(* IEC 61131-3 sources: pandora/pandora/aws-platform-main/aws-platform-main/src/Motion, 6 files *)

(* ---- Axis.st ---- *)
USING Esab.Utils.Assets;

NAMESPACE Esab.Motion

    /// Interface defining an axis.
    /// The interface supports both linear and rotary axes, defined through hardware configuration.
    INTERFACE IAxis
        METHOD PowerOn
        END_METHOD

        METHOD PowerOff
        END_METHOD

        METHOD Reset
            VAR_INPUT
                Restart : BOOL;
            END_VAR
        END_METHOD

        METHOD ExecutePositioningCommand : AxisCommandError
            VAR_INPUT
                command : AxisPositioningCommand;
            END_VAR
        END_METHOD

        METHOD ExecuteHomingCommand : AxisCommandError
            VAR_INPUT
                command: AxisHomingCommand;
            END_VAR
        END_METHOD

        METHOD InvalidateHoming
        END_METHOD

        METHOD Halt
        END_METHOD

        METHOD SetJogSpeed
            VAR_INPUT
                value : LREAL;
            END_VAR
        END_METHOD

        METHOD SetJogHighSpeed
            VAR_INPUT
                value : LREAL;
            END_VAR
        END_METHOD

        METHOD SetObjectRadius
            VAR_INPUT
                value : LREAL;
            END_VAR
        END_METHOD

        METHOD JogPositive
            VAR_INPUT
                highSpeed : BOOL := FALSE;
            END_VAR
        END_METHOD

        METHOD JogNegative
            VAR_INPUT
                highSpeed : BOOL := FALSE;
            END_VAR
        END_METHOD

        METHOD IsEnabled : BOOL
        END_METHOD

        METHOD IsBusy : BOOL
        END_METHOD

        METHOD IsHomed : BOOL
        END_METHOD

        METHOD HasError : BOOL
        END_METHOD

        METHOD AtStandstill : BOOL
        END_METHOD

        METHOD ActualLinearPosition : LREAL
        END_METHOD

        METHOD ActualLinearVelocity : LREAL
        END_METHOD

        METHOD ActualAngularPosition : LREAL
        END_METHOD

        METHOD ActualAngularVelocity : LREAL
        END_METHOD
    END_INTERFACE

    TYPE
        AxisCommandError : INT(
            NoError := 0,
            UnsupportedCommandType := 1,
            UnsupportedHomingType := 2,
            AxisNotEnabled := 3
        ) := AxisCommandError#NoError;

        AxisPositioningCommand : STRUCT
            CommandType : AxisCommandType := AxisCommandType#Absolute;
            /// NOTE: Only modulo axes supports setting the mode.
            PositioningDirection : AxisPositioningDirection := AxisPositioningDirection#Nearest;
            Id : INT := 0;
            Position : LREAL := 0.0;
            Velocity : LREAL := -1.0;
            Acceleration : LREAL := -1.0;
            Deceleration : LREAL := -1.0;
            Jerk : LREAL := -1.0;
        END_STRUCT;

        AxisCommandType : INT(
            Invalid     := -1,
            Absolute    := 0,
            Relative    := 1,
            Velocity    := 2,
            Halt        := 3
        ) := AxisCommandType#Invalid;

        AxisPositioningDirection : INT(
            Nearest := 0,
            Positive := 1,
            Negative := 2
        ) := AxisPositioningDirection#Nearest;

        AxisHomingCommand : STRUCT
            HomingType : AxisHomingType := AxisHomingType#DirectAbsolute;
            Position : LREAL := 0.0;
        END_STRUCT;

        AxisHomingType : INT(
            Invalid := -1,
            DirectAbsolute := 0,
            DirectRelative := 1,
            Active := 2,
            Passive := 3,
            AbsoluteEncoderAdjustementRelative := 4,
            AbsoluteEncoderAdjustementAbsolute := 5
        ) := AxisHomingType#Invalid;

        AxisState : INT(
            Enabled := 0,
            Disabled := 1,
            Error := 2,
            Homing := 3,
            Moving := 4
        ) := AxisState#Disabled;

        AxisType : INT(
            Linear := 0,
            Rotary := 1
        ) := AxisType#Rotary;

        AxisRuntimeParameters : STRUCT
            JogSpeed : LREAL := 10.0;
            JogHighSpeed : LREAL := 20.0;
            ObjectRadius : LREAL := 1500.0;
        END_STRUCT;

        AxisHardwareConfiguration : STRUCT
            AxisType : AxisType := AxisType#Linear;
        END_STRUCT;
    END_TYPE

    CLASS AxisObservable IMPLEMENTS IAssetObservable
        VAR PUBLIC
            State : AxisState;
            Enabled : BOOL;
            Accelerating : BOOL;
            Decelerating : BOOL;
            Standstill : BOOL;
            Homed : BOOL;
            Error : BOOL;
            ErrorId : WORD;
            Busy : BOOL;
            Done : BOOL;
            LatestCommandId : INT;
            LinearPosition : LREAL;
            LinearVelocity : LREAL;
            AngularPosition : LREAL;
            AngularVelocity : LREAL;
            ObjectRadius : LREAL;
        END_VAR
    END_CLASS

END_NAMESPACE

(* ---- WeldHeadManipulator.st ---- *)
USING Esab.Hmi.Modules;
USING Esab.Utils.Assets;
USING Esab.Utils.Alarming;
USING System.FastMath;

NAMESPACE Esab.Motion

    INTERFACE IWeldHeadManipulator
        METHOD Enable : WeldHeadManipulatorErrorCode
        END_METHOD

        METHOD Disable
        END_METHOD

        /// Interpolated motion, axes will arrive at the same time
        METHOD Move : WeldHeadManipulatorErrorCode
            VAR_INPUT
                position : ARRAY [0..1] OF LREAL := [0.0, 0.0];
                speed : LREAL := -1;
            END_VAR
        END_METHOD

        /// Non-interpolated movement
        METHOD Move : WeldHeadManipulatorErrorCode
            VAR_INPUT
                position : ARRAY [0..1] OF LREAL := [0.0, 0.0];
                speed : ARRAY [0..1] OF LREAL := [-1.0, -1.0];
            END_VAR
        END_METHOD

        METHOD IsEnabled : BOOL
        END_METHOD

        METHOD GetPosition : ARRAY [0..1] OF LREAL
        END_METHOD

        METHOD GetSpeed : LREAL
        END_METHOD

        METHOD GetVelocity : ARRAY [0..1] OF LREAL
        END_METHOD

        METHOD GetControlMode : WeldHeadManipulatorControlMode
        END_METHOD

        METHOD SetControlMode
            VAR_INPUT
                controlMode : WeldHeadManipulatorControlMode;
            END_VAR
        END_METHOD
    END_INTERFACE

    /// Class that wraps all axes that are used to manipulate the welding head.
    /// Depending on the hardware configuration this may include:
    /// - Horizontal slide axis
    /// - Vertical slide axis
    /// - Tilt (Not implemented)
    /// - Clock position slide (Not implemented)
    CLASS WeldHeadManipulator EXTENDS Asset IMPLEMENTS IAssetRequester, IWeldHeadManipulator, IPositionChangedListener
        VAR PRIVATE
            _runtimeParameters : REF_TO WeldHeadManipulatorRuntimeParameters;
            _hardwareConfiguration : REF_TO WeldHeadManipulatorHardwareConfiguration;
            _assetsManager : IAssetsManager;

            _horizontalSlide : IAxis;
            _verticalSlide : IAxis;

            _horizontalSlideObservable : REF_TO AxisObservable;
            _verticalSlideObservable : REF_TO AxisObservable;

            _horizontalSlideCommand : Esab.Motion.AxisPositioningCommand;
            _verticalSlideCommand : Esab.Motion.AxisPositioningCommand;

            _currentJogDirection : JoystickPosition := JoystickPosition#None;
            _motionJoystick : IJoystick := NULL;
        END_VAR

        METHOD PUBLIC Setup
            VAR_INPUT
                runtimeParameters : REF_TO WeldHeadManipulatorRuntimeParameters;
                hardwareConfiguration : REF_TO WeldHeadManipulatorHardwareConfiguration;
                assetsManager : IAssetsManager;
                setupAlarm : IAlarm;
            END_VAR

            _runtimeParameters := runtimeParameters;
            _hardwareConfiguration := hardwareConfiguration;
            _assetsManager := assetsManager;

            _isSetup := _runtimeParameters <> NULL AND _hardwareConfiguration <> NULL AND _assetsManager <> NULL;
        END_METHOD

        METHOD PUBLIC OVERRIDE Execute
            SUPER.Execute();

            IF _setupAlarm.IsActive() THEN
                RETURN;
            END_IF;

            THIS.RequestMotionJoystick();

            IF _horizontalSlideObservable = NULL THEN
                _horizontalSlideObservable ?= _assetsManager.ObserveAsset(Esab.AssetIdentifier#HorizontalSlideAxis);
            END_IF;

            IF _verticalSlideObservable = NULL THEN
                _verticalSlideObservable ?= _assetsManager.ObserveAsset(Esab.AssetIdentifier#VerticalSlideAxis);
            END_IF;

            IF _runtimeParameters^.controlMode = WeldHeadManipulatorControlMode#JoystickJog THEN
                THIS.HandleSlideJog();
            END_IF;
        END_METHOD

        METHOD PUBLIC Enable : WeldHeadManipulatorErrorCode
            VAR_TEMP
                currentPosition : ARRAY [0..1] OF LREAL;
            END_VAR

            IF NOT THIS.RequestAndLockAxis() THEN
                Enable := WeldHeadManipulatorErrorCode#AssetsNotAvailable;
                RETURN;
            END_IF;

            IF NOT _horizontalSlide.IsEnabled() THEN
                _horizontalSlide.PowerOn();
            END_IF;

            IF NOT _verticalSlide.IsEnabled() THEN
                _verticalSlide.PowerOn();
            END_IF;

            IF _horizontalSlide.HasError() OR _verticalSlide.HasError() THEN
                Enable := WeldHeadManipulatorErrorCode#AxisError;
                RETURN;
            END_IF;

            currentPosition[0] := _horizontalSlide.ActualLinearPosition();
            currentPosition[1] := _verticalSlide.ActualLinearPosition();

            THIS.Move(currentPosition, -1.0);
        END_METHOD

        METHOD PUBLIC Disable
            IF _horizontalSlide <> NULL THEN
                _horizontalSlide.Halt();
            END_IF;

            IF _verticalSlide <> NULL THEN
                _verticalSlide.Halt();
            END_IF;

            THIS.UnlockAxis();
        END_METHOD

        METHOD PUBLIC Move : WeldHeadManipulatorErrorCode
            VAR_INPUT
                position : ARRAY [0..1] OF LREAL := [0.0, 0.0];
                speed : LREAL := -1;
            END_VAR

            VAR_TEMP
                speedComponents : ARRAY [0..1] OF LREAL;
                currentPosition : ARRAY [0..1] OF LREAL;
            END_VAR

            IF _horizontalSlide = NULL OR _verticalSlide = NULL THEN
                Move := WeldHeadManipulatorErrorCode#AssetsNotAvailable;
                RETURN;
            END_IF;

            IF _horizontalSlide.HasError() OR _verticalSlide.HasError() THEN
                Move := WeldHeadManipulatorErrorCode#AxisError;
                RETURN;
            END_IF;

            currentPosition[0] := _horizontalSlide.ActualLinearPosition();
            currentPosition[1] := _verticalSlide.ActualLinearPosition();

            IF speed > 1.0 THEN
                speedComponents := THIS.CalculateSpeed(speed, currentPosition, position);
            ELSIF speed < 0.0 THEN
                speedComponents := THIS.CalculateSpeed(_runtimeParameters^.defaultSpeed, currentPosition, position);
            ELSE
                Move := WeldHeadManipulatorErrorCode#SpeedSetTooLow;
                RETURN;
            END_IF;

            _horizontalSlideCommand.CommandType := AxisCommandType#Absolute;
            _horizontalSlideCommand.Velocity := speedComponents[0];
            _horizontalSlideCommand.Position := position[0];

            _verticalSlideCommand.CommandType := AxisCommandType#Absolute;
            _verticalSlideCommand.Velocity := speedComponents[1];
            _verticalSlideCommand.Position := position[1];

            _horizontalSlide.ExecutePositioningCommand(_horizontalSlideCommand);
            _verticalSlide.ExecutePositioningCommand(_verticalSlideCommand);
        END_METHOD

        METHOD PUBLIC Move : WeldHeadManipulatorErrorCode
            VAR_INPUT
                position : ARRAY [0..1] OF LREAL := [0.0, 0.0];
                speed : ARRAY [0..1] OF LREAL := [-1.0, -1.0];
            END_VAR

            VAR_TEMP
                speedComponents : ARRAY [0..1] OF LREAL;
            END_VAR

            IF _horizontalSlide = NULL OR _verticalSlide = NULL THEN
                Move := WeldHeadManipulatorErrorCode#AssetsNotAvailable;
                RETURN;
            END_IF;

            IF _horizontalSlide.HasError() OR _verticalSlide.HasError() THEN
                Move := WeldHeadManipulatorErrorCode#AxisError;
                RETURN;
            END_IF;

            IF _runtimeParameters^.controlMode <> WeldHeadManipulatorControlMode#MoveToPosition THEN
                Move := WeldHeadManipulatorErrorCode#IncorrectControlMode;
                RETURN;
            END_IF;

            speedComponents := speed;

            _horizontalSlideCommand.CommandType := AxisCommandType#Absolute;
            _horizontalSlideCommand.Velocity := speedComponents[0];
            _horizontalSlideCommand.Position := position[0];

            _verticalSlideCommand.CommandType := AxisCommandType#Absolute;
            _verticalSlideCommand.Velocity := speedComponents[1];
            _verticalSlideCommand.Position := position[1];

            _horizontalSlide.ExecutePositioningCommand(_horizontalSlideCommand);
            _verticalSlide.ExecutePositioningCommand(_verticalSlideCommand);
        END_METHOD

        METHOD PUBLIC IsEnabled : BOOL
            IF THIS.InControl() THEN
                IsEnabled := _horizontalSlide.IsEnabled() AND _verticalSlide.IsEnabled();
            ELSE
                IsEnabled := FALSE;
            END_IF;
        END_METHOD

        METHOD PUBLIC GetPosition : ARRAY [0..1] OF LREAL
            IF _horizontalSlideObservable <> NULL AND _verticalSlideObservable <> NULL THEN
                GetPosition[0] := _horizontalSlideObservable^.LinearPosition;
                GetPosition[1] := _verticalSlideObservable^.LinearPosition;
            END_IF;
        END_METHOD

        METHOD PUBLIC GetSpeed : LREAL
            IF _horizontalSlideObservable <> NULL AND _verticalSlideObservable <> NULL THEN
                GetSpeed := Sqrt(_horizontalSlideObservable^.LinearVelocity * _horizontalSlideObservable^.LinearVelocity +
                                 _verticalSlideObservable^.LinearVelocity * _verticalSlideObservable^.LinearVelocity);
            END_IF;
        END_METHOD

        METHOD PUBLIC GetVelocity : ARRAY [0..1] OF LREAL
            IF _horizontalSlideObservable <> NULL AND _verticalSlideObservable <> NULL THEN
                GetVelocity[0] := _horizontalSlideObservable^.LinearVelocity;
                GetVelocity[1] := _verticalSlideObservable^.LinearVelocity;
            END_IF;
        END_METHOD

        METHOD PUBLIC GetControlMode : WeldHeadManipulatorControlMode
            GetControlMode := _runtimeParameters^.controlMode;
        END_METHOD

        METHOD PUBLIC SetControlMode
            VAR_INPUT
                controlMode : WeldHeadManipulatorControlMode;
            END_VAR;

            IF controlMode <> WeldHeadManipulatorControlMode#JoystickJog THEN
                _currentJogDirection := JoystickPosition#None;
            END_IF;

            _runtimeParameters^.controlMode := controlMode;
        END_METHOD

        METHOD PUBLIC AssetAssigned
            VAR_INPUT
                asset : REF_TO Esab.Utils.Assets.Asset;
            END_VAR

            ;
        END_METHOD

        METHOD PUBLIC AssetRemoved
            VAR_INPUT
                identifier : INT;
            END_VAR

            ;
        END_METHOD

        METHOD PUBLIC OVERRIDE Observe : IAssetObservable
            ;
        END_METHOD

        METHOD PRIVATE RequestAndLockAxis : BOOL
            VAR_TEMP
                success : BOOL := TRUE;
                asset : REF_TO Asset := NULL;
            END_VAR

            IF _hardwareConfiguration^.horizontalSlideAxis AND _horizontalSlide = NULL THEN
                asset := _assetsManager.RequestAssetHandle(THIS, Esab.AssetIdentifier#HorizontalSlideAxis);
                IF asset <> NULL THEN
                    _horizontalSlide ?= asset^;
                ELSE
                    success := FALSE;
                END_IF;
            END_IF;

            IF _hardwareConfiguration^.verticalSlideAxis AND _verticalSlide = NULL THEN
                asset := _assetsManager.RequestAssetHandle(THIS, Esab.AssetIdentifier#VerticalSlideAxis);
                IF asset <> NULL THEN
                    _verticalSlide ?= asset^;
                ELSE
                    success := FALSE;
                END_IF;
            END_IF;

            IF success THEN
                IF _horizontalSlide <> NULL THEN
                    asset ?= _horizontalSlide;
                    asset^.Lock();
                END_IF;

                IF _verticalSlide <> NULL THEN
                    asset ?= _verticalSlide;
                    asset^.Lock();
                END_IF;
            END_IF;

            RequestAndLockAxis := success;
        END_METHOD

        METHOD PRIVATE InControl : BOOL
            VAR_TEMP
                asset : REF_TO asset;
            END_VAR

            InControl := TRUE;

            IF _horizontalSlide <> NULL THEN
                asset ?= _horizontalSlide;
                IF NOT asset^.IsLocked() THEN
                    InControl := FALSE;
                END_IF;
            ELSE
                InControl := FALSE;
            END_IF;

            IF _verticalSlide <> NULL THEN
                asset ?= _verticalSlide;
                IF NOT asset^.IsLocked() THEN
                    InControl := FALSE;
                END_IF;
            ELSE
                InControl := FALSE;
            END_IF;
        END_METHOD

        METHOD PRIVATE UnlockAxis
            VAR_TEMP
                asset : REF_TO Asset;
            END_VAR

            IF _horizontalSlide <> NULL THEN
                asset ?= _horizontalSlide;
                asset^.Unlock();
            END_IF;

            IF _verticalSlide <> NULL THEN
                asset ?= _verticalSlide;
                asset^.Unlock();
            END_IF;
        END_METHOD

        METHOD PRIVATE CalculateSpeed : ARRAY [0..1] OF LREAL
            VAR_INPUT
                speed : LREAL;
                currentPosition : ARRAY [0..1] OF LREAL;
                targetPosition : ARRAY [0..1] OF LREAL;
            END_VAR

            VAR_TEMP
                theta : LREAL;
                distance : ARRAY [0..1] OF LREAL;
            END_VAR

            distance[0] := Abs(targetPosition[0]-currentPosition[0]);
            distance[1] := Abs(targetPosition[1]-currentPosition[1]);

            theta := ATan(distance[1] / distance[0]);

            CalculateSpeed[0] := speed * Cos(theta);
            CalculateSpeed[1] := speed * Sin(theta);

            IF CalculateSpeed[0] < 1.0 THEN
                CalculateSpeed[0] := 1.0;
            END_IF;

            IF CalculateSpeed[1] < 1.0 THEN
                CalculateSpeed[1] := 1.0;
            END_IF;
        END_METHOD

        METHOD PUBLIC OnPositionChanged
            VAR_INPUT
                position : JoystickPosition;
            END_VAR
                IF _runtimeParameters^.controlMode <> WeldHeadManipulatorControlMode#JoystickJog THEN
                    RETURN;
                END_IF;

                _currentJogDirection := position;
        END_METHOD

        METHOD PRIVATE HandleSlideJog
            IF _horizontalSlide = NULL OR _verticalSlide = NULL THEN
                RETURN;
            END_IF;

            IF _horizontalSlide.HasError() OR _verticalSlide.HasError() THEN
                RETURN;
            END_IF;

            CASE _currentJogDirection OF
                JoystickPosition#None:
                    _horizontalSlide.Halt();
                    _verticalSlide.Halt();
                JoystickPosition#Center:
                    _horizontalSlide.Halt();
                    _verticalSlide.Halt();
                JoystickPosition#Up:
                    _horizontalSlide.Halt();
                    _verticalSlide.JogPositive();
                JoystickPosition#Down:
                    _horizontalSlide.Halt();
                    _verticalSlide.JogNegative();
                JoystickPosition#Square:
                    _horizontalSlide.JogPositive();
                    _verticalSlide.Halt();
                JoystickPosition#Triangle:
                    _horizontalSlide.JogNegative();
                    _verticalSlide.Halt();
            END_CASE;
        END_METHOD

        METHOD PRIVATE RequestMotionJoystick
            VAR_TEMP
                assetHandle : REF_TO Asset;
            END_VAR

            IF _motionJoystick = NULL THEN
                assetHandle := THIS._assetsManager.RequestAssetHandle(THIS, Esab.AssetIdentifier#P_Joystick_MotionJoystick);

                IF assetHandle <> NULL THEN
                    _motionJoystick ?= assetHandle^;
                    IF _motionJoystick <> NULL THEN
                        _motionJoystick.SetPositionChangedListener(THIS);
                    END_IF;
                END_IF;
            END_IF;
        END_METHOD

    END_CLASS

    TYPE
        WeldHeadManipulatorRuntimeParameters : STRUCT
        /// Speed used when move command speed < 0.0
            defaultSpeed : LREAL := 10.0;
            controlMode : WeldHeadManipulatorControlMode;
        END_STRUCT;

        WeldHeadManipulatorHardwareConfiguration : STRUCT
            /// X-axis
            horizontalSlideAxis : BOOL := TRUE;
            /// Z-axis
            verticalSlideAxis : BOOL := TRUE;
        END_STRUCT;

        WeldHeadManipulatorErrorCode : INT(
            NoError := 0,
            AssetsNotAvailable := 1,
            AxisError := 2,
            SpeedSetTooLow := 3,
            IncorrectControlMode := 4
        ) := WeldHeadManipulatorErrorCode#NoError;

        WeldHeadManipulatorControlMode : INT(
            NoControl := 0,
            JoystickJog := 1,
            MoveToPosition := 2
        ) := WeldHeadManipulatorControlMode#NoControl;
    END_TYPE
END_NAMESPACE

(* ---- AnalogAxis.st ---- *)
USING Esab.Motion.MeasurementSystem;
USING Esab.Utils.Assets;
USING Esab.Utils.Timer;
USING Esab.Utils.Alarming;
USING Esab.Io;

USING System.FastMath;

NAMESPACE Esab.Motion

    /// Implements an axis with the following properties:
    ///     - The axis is controlled via digital and analog I/O:
    ///         - Forwards/positive direction (digital out)
    ///         - Backwards/negative direction (digital out)
    ///         - Speed (analog out)
    /// To measure the position (if applicable) a measurement system should
    /// be provided. The axis will work "fine" without it but it will be limited to
    /// speed control without feedback.
    CLASS AnalogAxis EXTENDS Asset IMPLEMENTS IAxis, IMeasurementSystemListener
        VAR PRIVATE
            _io : REF_TO AnalogAxisIo;
            _runtimeParameters : REF_TO AnalogAxisRuntimeParameters;
            _hardwareConfiguration : REF_TO AnalogAxisHardwareConfiguration;
            _measurementSystem : IMeasurementSystem1D;
            _speedMeasurementTimer : ITimer;
            _speedMonitoringAlarm : IAlarm;

            _observable : AxisObservable;

            _setVelocity : LREAL := 0.0;
            _jogPositive : BOOL := FALSE;
            _jogNegative : BOOL := FALSE;
            _highSpeed : BOOL := FALSE;
            _isJogging : BOOL := FALSE;
            _isHomed : BOOL := FALSE;
            _poweredOn : BOOL := FALSE;
            _measuring : BOOL := FALSE;
            _hasPassedReferencePointOnce : BOOL := FALSE;
        END_VAR

        METHOD PUBLIC Setup
            VAR_INPUT
                io : REF_TO AnalogAxisIo;
                runtimeParameters : REF_TO AnalogAxisRuntimeParameters;
                hardwareConfiguration : REF_TO AnalogAxisHardwareConfiguration;
                measurementSystem : IMeasurementSystem1D;
                speedMeasurementTimer : ITimer;
                speedMonitoringAlarm : IAlarm;
                setupAlarm : IAlarm;
            END_VAR

            _io := io;
            _runtimeParameters := runtimeParameters;
            _hardwareConfiguration := hardwareConfiguration;
            _measurementSystem := measurementSystem;
            _speedMeasurementTimer := speedMeasurementTimer;
            _speedMonitoringAlarm := speedMonitoringAlarm;
            _setupAlarm := setupAlarm;

            _isSetup := _io <> NULL AND
                        _hardwareConfiguration <> NULL AND
                        _runtimeParameters <> NULL AND
                        _measurementSystem <> NULL AND
                        _speedMonitoringAlarm <> NULL;

            IF _isSetup THEN
                _measurementSystem.SetListener(THIS);
            END_IF;
        END_METHOD

        METHOD PUBLIC OVERRIDE Execute
            VAR_TEMP
                _actualSpeedInMmPerS : LREAL;
                _speedPercentage : LREAL;
            END_VAR

            SUPER.Execute();

            IF _setupAlarm.IsActive() THEN
                RETURN;
            END_IF;

            _measurementSystem.Execute();

            _speedMeasurementTimer.Execute(_measuring, _runtimeParameters^.SpeedSettlingTime);

            IF _measuring THEN
                IF _speedMeasurementTimer.Expired() THEN
                    THIS.AdjustMaxSpeed();
                    _measuring := FALSE;
                END_IF;
            ELSE
                IF _isJogging OR _jogPositive OR _jogNegative THEN
                    IF NOT _isJogging AND (_jogPositive OR _jogNegative) THEN
                        IF _jogPositive THEN
                            IF _highSpeed THEN
                                THIS.SetVelocity(_runtimeParameters^.Axis.JogHighSpeed);
                            ELSE
                                THIS.SetVelocity(_runtimeParameters^.Axis.JogSpeed);
                            END_IF;
                        ELSIF _jogNegative THEN
                            IF _highSpeed THEN
                                THIS.SetVelocity(-_runtimeParameters^.Axis.JogHighSpeed);
                            ELSE
                                THIS.SetVelocity(-_runtimeParameters^.Axis.JogSpeed);
                            END_IF;
                        END_IF;

                        _isJogging := TRUE;
                    END_IF;

                    IF _isJogging AND NOT (_jogPositive OR _jogNegative) THEN
                        THIS.Halt();
                        _isJogging := FALSE;
                    END_IF;
                END_IF;
            END_IF;

            _jogPositive := FALSE;
            _jogNegative := FALSE;
            _highSpeed := FALSE;

            _speedMonitoringAlarm.Execute(NOT THIS.AtStandstill() AND ABS(THIS.ActualLinearVelocity() - _setVelocity) > 0.05);

            THIS.UpdateState();
            THIS.UpdateObservable();
        END_METHOD

        METHOD PUBLIC PowerOn
            _poweredOn := TRUE;
            _io^.Outputs.RemoteControl.Set();
        END_METHOD

        METHOD PUBLIC PowerOff
            _poweredOn := FALSE;
            _io^.Outputs.RemoteControl.Reset();
        END_METHOD

        METHOD PUBLIC Reset
            VAR_INPUT
                Restart : BOOL;
            END_VAR

            ;
        END_METHOD

        METHOD PUBLIC ExecutePositioningCommand : AxisCommandError
            VAR_INPUT
                command : AxisPositioningCommand;
            END_VAR

            VAR_TEMP
                _error : AxisCommandError := AxisCommandError#NoError;
            END_VAR

            IF NOT THIS.IsEnabled() THEN
                ExecutePositioningCommand := AxisCommandError#AxisNotEnabled;
                RETURN;
            END_IF;

            CASE command.CommandType OF
                AxisCommandType#Velocity:
                    THIS.SetVelocity(command.Velocity);
                AxisCommandType#Halt:
                    THIS.SetVelocity(0.0);
            ELSE
                _error := AxisCommandError#UnsupportedCommandType;
            END_CASE;

            ExecutePositioningCommand := _error;
        END_METHOD

        METHOD PUBLIC ExecuteHomingCommand : AxisCommandError
            VAR_INPUT
                command : AxisHomingCommand;
            END_VAR

            VAR_TEMP
                _error : AxisCommandError := AxisCommandError#NoError;
            END_VAR

            IF NOT THIS.IsEnabled() THEN
                ExecuteHomingCommand := AxisCommandError#AxisNotEnabled;
                RETURN;
            END_IF;

            CASE command.HomingType OF
                AxisHomingType#Active:
                    THIS.SetVelocity(_runtimeParameters^.MeasuringSpeed);
                    _measuring := TRUE;
            END_CASE;

            ExecuteHomingCommand := _error;
        END_METHOD

        METHOD PUBLIC InvalidateHoming
            _isHomed := FALSE;
            _hasPassedReferencePointOnce := FALSE;
        END_METHOD

        METHOD PUBLIC Halt
            _jogNegative := FALSE;
            _jogPositive := FALSE;
            _isJogging := FALSE;

            THIS.SetVelocity(0.0);
        END_METHOD

        METHOD PUBLIC SetJogSpeed
            VAR_INPUT
                value : LREAL;
            END_VAR

            _runtimeParameters^.Axis.JogSpeed := value;
        END_METHOD

        METHOD PUBLIC SetJogHighSpeed
            VAR_INPUT
                value : LREAL;
            END_VAR

            _runtimeParameters^.Axis.JogHighSpeed := value;
        END_METHOD

        METHOD PUBLIC SetObjectRadius
            VAR_INPUT
                value : LREAL;
            END_VAR

            _runtimeParameters^.Axis.ObjectRadius := value;
        END_METHOD

        METHOD PUBLIC JogPositive
            VAR_INPUT
                highSpeed : BOOL := FALSE;
            END_VAR

            IF NOT THIS.IsEnabled() THEN
                RETURN;
            END_IF;

            _highSpeed := highSpeed;
            _jogPositive := TRUE;
            _jogNegative := FALSE;
        END_METHOD

        METHOD PUBLIC JogNegative
            VAR_INPUT
                highSpeed : BOOL := FALSE;
            END_VAR

            IF NOT THIS.IsEnabled() THEN
                RETURN;
            END_IF;

            _highSpeed := highSpeed;
            _jogPositive := FALSE;
            _jogNegative := TRUE;
        END_METHOD

        METHOD PUBLIC IsEnabled : BOOL
            IsEnabled := _poweredOn;
        END_METHOD

        METHOD PUBLIC IsBusy : BOOL
            IsBusy := NOT THIS.AtStandstill();
        END_METHOD

        METHOD PUBLIC HasError : BOOL
            HasError := THIS._speedMonitoringAlarm.IsActive() OR THIS._setupAlarm.IsActive();
        END_METHOD

        METHOD PUBLIC AtStandstill : BOOL
            AtStandstill := ABS(THIS.ActualLinearVelocity()) < 0.5;
        END_METHOD

        METHOD PUBLIC IsHomed : BOOL
            IsHomed := _isHomed;
        END_METHOD

        METHOD PUBLIC ActualLinearPosition : LREAL
            ActualLinearPosition := _measurementSystem.GetMeasuredPosition();
        END_METHOD

        METHOD PUBLIC ActualLinearVelocity : LREAL
            ActualLinearVelocity := _measurementSystem.GetMeasuredVelocity();
        END_METHOD

        METHOD PUBLIC ActualAngularPosition : LREAL
            VAR_TEMP
                _position : LREAL := 0.0;
            END_VAR

            IF _hardwareConfiguration^.Axis.AxisType = AxisType#Rotary THEN
                _position := _measurementSystem.GetMeasuredPosition() / (2 * Constants#PI * _runtimeParameters^.Axis.ObjectRadius) * 360.0;
            END_IF;

            ActualAngularPosition := _position;
        END_METHOD

        METHOD PUBLIC ActualAngularVelocity : LREAL
            VAR_TEMP
                _velocity : LREAL := 0.0;
            END_VAR

            IF _hardwareConfiguration^.Axis.AxisType = AxisType#Rotary THEN
                _velocity := _measurementSystem.GetMeasuredVelocity() / (2 * Constants#PI * _runtimeParameters^.Axis.ObjectRadius) * 360.0;
            END_IF;

            ActualAngularVelocity := _velocity;
        END_METHOD

        METHOD PUBLIC OVERRIDE Observe : IAssetObservable
            Observe := _observable;
        END_METHOD

        METHOD PUBLIC ArrivedAtReferencePoint
            IF _hasPassedReferencePointOnce THEN
                THIS.SetRadiusFromCircumference(_measurementSystem.GetMeasuredPosition());
                _isHomed := TRUE;
            ELSE
                _hasPassedReferencePointOnce := TRUE;
            END_IF;

            _measurementSystem.ResetMeasuredPosition();
        END_METHOD

        METHOD PRIVATE SetRadiusFromCircumference
            VAR_INPUT
                circumference : LREAL;
            END_VAR

            _runtimeParameters^.Axis.ObjectRadius := circumference / (2 * Constants#PI);
        END_METHOD

        METHOD PRIVATE UpdateObservable
            _observable.State := THIS.GetState();
            _observable.Enabled := THIS.IsEnabled();
            _observable.Accelerating := FALSE;
            _observable.Decelerating := FALSE;
            _observable.Standstill := THIS.AtStandstill();
            _observable.Homed := THIS.IsHomed();
            _observable.Error := THIS.HasError();
            _observable.ErrorId := WORD#16#0000;
            _observable.Busy := THIS.IsBusy();
            _observable.Done := FALSE;
            _observable.LatestCommandId := 16#0000;
            _observable.LinearPosition := THIS.ActualLinearPosition();
            _observable.LinearVelocity := THIS.ActualLinearVelocity();
            _observable.AngularPosition := THIS.ActualAngularPosition();
            _observable.AngularVelocity := THIS.ActualAngularVelocity();
        END_METHOD

        METHOD PRIVATE UpdateState
            IF THIS.HasError() THEN
                _currentState := AxisState#Error;
            ELSIF THIS.IsBusy() THEN
                _currentState := AxisState#Moving;
            ELSIF THIS.IsEnabled() THEN
                _currentState := AxisState#Enabled;
            ELSE
                _currentState := AxisState#Disabled;
            END_IF;
        END_METHOD

        METHOD PRIVATE SetVelocity
            VAR_INPUT
                velocity : LREAL;
            END_VAR

            VAR_TEMP
                speed : REAL;
            END_VAR

            _setVelocity := velocity;

            speed := TO_REAL(ABS(velocity) / _hardwareConfiguration^.MaximumSpeed);

            IF velocity > 0.01 THEN
                _io^.Outputs.SpeedReference.SetValue(speed);
                _io^.Outputs.Forward.Set();
                _io^.Outputs.Reverse.Reset();
            ELSIF velocity < -0.01 THEN
                _io^.Outputs.SpeedReference.SetValue(speed);
                _io^.Outputs.Forward.Reset();
                _io^.Outputs.Reverse.Set();
            ELSE
                _io^.Outputs.SpeedReference.SetValue(REAL#0.0);
                _io^.Outputs.Forward.Reset();
                _io^.Outputs.Reverse.Reset();
            END_IF;
        END_METHOD

        METHOD PRIVATE AdjustMaxSpeed
            _hardwareConfiguration^.MaximumSpeed := _measurementSystem.GetMeasuredVelocity() / _setVelocity * _hardwareConfiguration^.MaximumSpeed;
            // We also need to update the outputs when we adjust the max speed
            THIS.SetVelocity(_setVelocity);
        END_METHOD
    END_CLASS

    TYPE
        AnalogAxisRuntimeParameters : STRUCT
            Axis : AxisRuntimeParameters;
            MeasuringSpeed : LREAL := 8.33;
            SpeedSettlingTime : LTIME := LT#5s;
        END_STRUCT;

        AnalogAxisHardwareConfiguration : STRUCT
            Axis : AxisHardwareConfiguration;
            MaximumSpeed : LREAL := 100.0;
        END_STRUCT;
    END_TYPE

    TYPE
        AnalogAxisIo : STRUCT
            Inputs : AnalogAxisInputs;
            Outputs : AnalogAxisOutputs;
        END_STRUCT;

        AnalogAxisInputs : STRUCT
            Error : DigitalInput;
        END_STRUCT;

        AnalogAxisOutputs : STRUCT
            Forward : DigitalOutput;
            Reverse : DigitalOutput;
            RemoteControl : DigitalOutput;
            SpeedReference : RealNormalizedOutput;
        END_STRUCT;
    END_TYPE

END_NAMESPACE

(* ---- SimulatedAnalogAxis.st ---- *)
USING Esab.Utils.Assets;
USING Esab.Utils.Alarming;

USING System.Timer;
USING System.FastMath;

NAMESPACE Esab.Motion

    CLASS SimulatedAnalogAxis EXTENDS Asset IMPLEMENTS IAxis
        VAR PRIVATE
            _runtimeParameters : REF_TO AnalogAxisRuntimeParameters;
            _hardwareConfiguration : REF_TO AnalogAxisHardwareConfiguration;
            _observable : AxisObservable;
            _lastRuntime : LTIME;
            _runtime : LTIME;
            _runtimeTimer : TimeAccumulator;
            _poweredOn : BOOL;
            _velocity : LREAL;
            _position : LREAL;
            _isJogging : BOOL;
            _isHomed : BOOL;
            _jogPositive : BOOL;
            _jogNegative : BOOL;
            _highSpeed : BOOL;
        END_VAR

        METHOD PUBLIC Setup
            VAR_INPUT
                runtimeParameters : REF_TO AnalogAxisRuntimeParameters;
                hardwareConfiguration : REF_TO AnalogAxisHardwareConfiguration;
                setupAlarm : IAlarm;
            END_VAR

            _runtimeParameters := runtimeParameters;
            _hardwareConfiguration := hardwareConfiguration;
            _setupAlarm := setupAlarm;

            _isSetup := _runtimeParameters <> NULL AND _hardwareConfiguration <> NULL;

            IF _isSetup THEN
                THIS.PowerOn();
            END_IF;
        END_METHOD

        METHOD PUBLIC OVERRIDE Execute
            VAR_TEMP
                moving : BOOL;
                passedTime : LREAL;
            END_VAR

            SUPER.Execute();

            IF _setupAlarm.IsActive() THEN
                RETURN;
            END_IF;

            _runtimeTimer(signal := NOT THIS.AtStandstill(), duration := LT#42d, reset := THIS.AtStandstill(), accumulatedTime => _runtime);

            passedTime := TO_LREAL(TO_LINT(_runtime))/1000.0;

            _position := _velocity * passedTime;

            IF _isJogging OR _jogPositive OR _jogNegative THEN
                IF NOT _isJogging AND (_jogPositive OR _jogNegative) THEN
                    IF _jogPositive THEN
                        IF _highSpeed THEN
                            THIS.SetVelocity(_runtimeParameters^.Axis.JogHighSpeed);
                        ELSE
                            THIS.SetVelocity(_runtimeParameters^.Axis.JogSpeed);
                        END_IF;
                    ELSIF _jogNegative THEN
                        IF _highSpeed THEN
                            THIS.SetVelocity(-_runtimeParameters^.Axis.JogHighSpeed);
                        ELSE
                            THIS.SetVelocity(-_runtimeParameters^.Axis.JogSpeed);
                        END_IF;
                    END_IF;

                    _isJogging := TRUE;
                END_IF;

                IF _isJogging AND NOT (_jogPositive OR _jogNegative) THEN
                    THIS.Halt();
                    _isJogging := FALSE;
                END_IF;
            END_IF;

            _jogPositive := FALSE;
            _jogNegative := FALSE;
            _highSpeed := FALSE;

            _lastRuntime := _runtime;

            THIS.UpdateObservable();
        END_METHOD

        METHOD PUBLIC PowerOn
            _poweredOn := TRUE;
        END_METHOD

        METHOD PUBLIC PowerOff
            _poweredOn := FALSE;
        END_METHOD

        METHOD PUBLIC Reset
            VAR_INPUT
                Restart : BOOL;
            END_VAR

            ;
        END_METHOD

        METHOD PUBLIC ExecutePositioningCommand : AxisCommandError
            VAR_INPUT
                command : AxisPositioningCommand;
            END_VAR

            VAR_TEMP
                _error : AxisCommandError := AxisCommandError#NoError;
            END_VAR

            IF NOT THIS.IsEnabled() THEN
                ExecutePositioningCommand := AxisCommandError#AxisNotEnabled;
                RETURN;
            END_IF;

            CASE command.CommandType OF
                AxisCommandType#Velocity:
                    THIS.SetVelocity(command.Velocity);
                AxisCommandType#Halt:
                    THIS.SetVelocity(0.0);
            ELSE
                _error := AxisCommandError#UnsupportedCommandType;
            END_CASE;

            ExecutePositioningCommand := _error;
        END_METHOD

        METHOD PUBLIC ExecuteHomingCommand : AxisCommandError
            VAR_INPUT
                command : AxisHomingCommand;
            END_VAR

            VAR_TEMP
                _error : AxisCommandError := AxisCommandError#NoError;
            END_VAR

            IF NOT THIS.IsEnabled() THEN
                ExecuteHomingCommand := AxisCommandError#AxisNotEnabled;
                RETURN;
            END_IF;

            ;
        END_METHOD

        METHOD PUBLIC InvalidateHoming
            _isHomed := FALSE;
        END_METHOD

        METHOD PUBLIC Halt
            THIS.SetVelocity(0.0);
        END_METHOD

        METHOD PUBLIC SetJogSpeed
            VAR_INPUT
                value : LREAL;
            END_VAR

            _runtimeParameters^.Axis.JogSpeed := value;
        END_METHOD

        METHOD PUBLIC SetJogHighSpeed
            VAR_INPUT
                value : LREAL;
            END_VAR

            _runtimeParameters^.Axis.JogHighSpeed := value;
        END_METHOD

        METHOD PUBLIC SetObjectRadius
            VAR_INPUT
                value : LREAL;
            END_VAR

            _runtimeParameters^.Axis.ObjectRadius := value;
        END_METHOD

        METHOD PUBLIC JogPositive
            VAR_INPUT
                highSpeed : BOOL := FALSE;
            END_VAR

            IF NOT THIS.IsEnabled() THEN
                RETURN;
            END_IF;

            _highSpeed := highSpeed;
            _jogPositive := TRUE;
            _jogNegative := FALSE;
        END_METHOD

        METHOD PUBLIC JogNegative
            VAR_INPUT
                highSpeed : BOOL := FALSE;
            END_VAR

            IF NOT THIS.IsEnabled() THEN
                RETURN;
            END_IF;

            _highSpeed := highSpeed;
            _jogPositive := FALSE;
            _jogNegative := TRUE;
        END_METHOD

        METHOD PUBLIC IsEnabled : BOOL
            IsEnabled := _poweredOn;
        END_METHOD

        METHOD PUBLIC IsBusy : BOOL
            IsBusy := Abs(_velocity) > 0.1;
        END_METHOD

        METHOD PUBLIC HasError : BOOL
            ;
        END_METHOD

        METHOD PUBLIC AtStandstill : BOOL
            AtStandstill := ABS(THIS.ActualLinearVelocity()) < 0.5;
        END_METHOD

        METHOD PUBLIC IsHomed : BOOL
            IsHomed := _isHomed;
        END_METHOD

        METHOD PUBLIC ActualLinearPosition : LREAL
            ActualLinearPosition := _position;
        END_METHOD

        METHOD PUBLIC ActualLinearVelocity : LREAL
            ActualLinearVelocity := _velocity;
        END_METHOD

        METHOD PUBLIC ActualAngularPosition : LREAL
            VAR_TEMP
                _angularPosition : LREAL := 0.0;
            END_VAR

            IF _hardwareConfiguration^.Axis.AxisType = AxisType#Rotary THEN
                _angularPosition := _position / (2 * Constants#PI * _runtimeParameters^.Axis.ObjectRadius) * 360.0;
            END_IF;

            ActualAngularPosition := _angularPosition;
        END_METHOD

        METHOD PUBLIC ActualAngularVelocity : LREAL
            VAR_TEMP
                _angularVelocity : LREAL := 0.0;
            END_VAR

            IF _hardwareConfiguration^.Axis.AxisType = AxisType#Rotary THEN
                _angularVelocity := _velocity / (2 * Constants#PI * _runtimeParameters^.Axis.ObjectRadius) * 360.0;
            END_IF;

            ActualAngularVelocity := _angularVelocity;
        END_METHOD

        METHOD PUBLIC OVERRIDE Observe : IAssetObservable
            Observe := _observable;
        END_METHOD

        METHOD PRIVATE SetVelocity
            VAR_INPUT
                velocity : LREAL;
            END_VAR

            _velocity := velocity;
        END_METHOD

        METHOD PRIVATE UpdateObservable
            _observable.Enabled := THIS.IsEnabled();
            _observable.Accelerating := FALSE;
            _observable.Decelerating := FALSE;
            _observable.Standstill := THIS.AtStandstill();
            _observable.Homed := THIS.IsHomed();
            _observable.Error := THIS.HasError();
            _observable.ErrorId := WORD#16#0000;
            _observable.Busy := THIS.IsBusy();
            _observable.Done := FALSE;
            _observable.LatestCommandId := 16#0000;
            _observable.LinearPosition := THIS.ActualLinearPosition();
            _observable.LinearVelocity := THIS.ActualLinearVelocity();
            _observable.AngularPosition := THIS.ActualAngularPosition();
            _observable.AngularVelocity := THIS.ActualAngularVelocity();
        END_METHOD
    END_CLASS

END_NAMESPACE

(* ---- TechnologyObjectAxis.st ---- *)
USING Esab.Utils.Assets;
USING Esab.Utils.Alarming;

USING Siemens.Simatic.S71500.MotionControl;
USING Siemens.Simatic.S71500.MotionControl.Native;

NAMESPACE Esab.Motion

    /// Implements a technology object position axis.
    /// This implementation depends on the Siemens TO object for motion.
    /// Currently does not support AxisType#Rotary.
    CLASS ToPosAxis EXTENDS Asset IMPLEMENTS IAxis
        VAR PRIVATE
            _axis : itfPosAxis := NULL;
            _runtimeParameters : REF_TO AxisRuntimeParameters;

            _latestAxisPositioningCommand : AxisPositioningCommand;
            _latestAxisHomingCommand : AxisHomingCommand;
            _latestCommand : itfCommand := NULL;
            _latestHomingCommand : itfHomeCommand := NULL;
            _jogPositive : BOOL := FALSE;
            _jogNegative : BOOL := FALSE;
            _jogUseHighSpeed : BOOL := FALSE;
            _observable : AxisObservable;
        END_VAR

        METHOD PUBLIC Setup
            VAR_INPUT
                axis : itfPosAxis;
                runtimeParameters : REF_TO AxisRuntimeParameters;
                setupAlarm : IAlarm;
            END_VAR

            _axis := axis;
            _runtimeParameters := runtimeParameters;
            _setupAlarm := setupAlarm;

            _isSetup := _axis <> NULL AND _runtimeParameters <> NULL;

            IF _isSetup AND NOT THIS.IsEnabled() THEN
                THIS.PowerOn();
            END_IF;
        END_METHOD

        METHOD PUBLIC OVERRIDE Execute
            SUPER.Execute();

            IF _setupAlarm.IsActive() THEN
                RETURN;
            END_IF;

            IF _jogUseHighSpeed THEN
                _axis.MoveJog(_jogPositive, _jogNegative, _runtimeParameters^.JogHighSpeed, -1.0, -1.0, -1.0, TRUE);
            ELSE
                _axis.MoveJog(_jogPositive, _jogNegative, _runtimeParameters^.JogSpeed, -1.0, -1.0, -1.0, TRUE);
            END_IF;

            _jogUseHighSpeed := FALSE;
            _jogPositive := FALSE;
            _jogNegative := FALSE;

            THIS.UpdateObservable();
        END_METHOD

        METHOD PUBLIC OVERRIDE UpdateState
            IF _setupAlarm.IsActive() THEN
                _currentState := AxisState#Error;
            ELSIF _axis.GetStatus().error THEN
                _currentState := AxisState#Error;
            ELSIF _latestHomingCommand <> NULL THEN
                _currentState := AxisState#Homing;
            ELSIF NOT _axis.GetStatus().standstill THEN
                _currentState := AxisState#Moving;
            ELSIF _axis.GetStatus().enable THEN
                _currentState := AxisState#Enabled;
            ELSE
                _currentState := AxisState#Disabled;
            END_IF;
        END_METHOD

        METHOD PUBLIC PowerOn
            _latestCommand := _axis.PowerOn(TRUE);
        END_METHOD

        METHOD PUBLIC PowerOff
            _latestCommand := _axis.PowerOff();
        END_METHOD

        METHOD PUBLIC Reset
            VAR_INPUT
                Restart : BOOL;
            END_VAR

            _latestAxisPositioningCommand.CommandType := AxisCommandType#Invalid;
            _latestCommand := NULL;
            _latestHomingCommand := NULL;

            _axis.ResetAlarms();

            IF Restart THEN
                _axis.Restart();
            END_IF;
        END_METHOD

        METHOD PUBLIC ExecutePositioningCommand : AxisCommandError
            VAR_INPUT
                command: AxisPositioningCommand;
            END_VAR

            CASE command.CommandType OF
                AxisCommandType#Absolute:
                    _latestCommand := _axis.MoveAbsolute(
                        Position := command.Position,
                        Velocity := command.Velocity,
                        Acceleration := command.Acceleration,
                        Deceleration := command.Deceleration,
                        Jerk := command.Jerk,
                        Direction := DirectionModulo#Positive
                    );
                AxisCommandType#Relative:
                    _latestCommand := _axis.MoveRelative(
                        Distance := command.Position,
                        Velocity := command.Velocity,
                        Acceleration := command.Acceleration,
                        Deceleration := command.Deceleration,
                        Jerk := command.Jerk
                    );
                AxisCommandType#Velocity:
                    _latestCommand := _axis.MoveVelocity(
                        Velocity := command.Velocity,
                        Acceleration := command.Acceleration,
                        Deceleration := command.Deceleration,
                        Jerk := command.Jerk,
                        Direction := Direction#VelocitySpecified,
                        PositionControlled := TRUE
                    );
                AxisCommandType#Halt:
                    _latestCommand := _axis.Halt(
                        Deceleration := command.Deceleration,
                        Jerk := command.Jerk
                    );
            END_CASE;

            //_invalidCommandAlarm(SIG := NOT (command.Type_ > AxisCommandType#Invalid AND
            //                                 command.Type_ < AxisCommandType#Last)
            //                    );

            _latestAxisPositioningCommand := command;
        END_METHOD

        METHOD PUBLIC ExecuteHomingCommand : AxisCommandError
            VAR_INPUT
                command: AxisHomingCommand;
            END_VAR

            CASE command.HomingType OF
                AxisHomingType#DirectAbsolute:
                    _latestHomingCommand := _axis.HomeDirect(command.Position, HomingModeDirect#ActualPositionAbsolute);
                AxisHomingType#DirectRelative:
                    _latestHomingCommand := _axis.HomeDirect(command.Position, HomingModeDirect#ActualPositionRelative);
                AxisHomingType#AbsoluteEncoderAdjustementAbsolute:
                    _latestHomingCommand := _axis.HomeAbsEncoder(command.Position, HomingModeAbsEncoder#AdjustmentSensorAbsolute);
            END_CASE;
        END_METHOD

        METHOD PUBLIC InvalidateHoming
            ;
        END_METHOD

        METHOD PUBLIC Halt
            _latestCommand := _axis.Halt();
        END_METHOD

        METHOD PUBLIC SetJogSpeed
            VAR_INPUT
                value : LREAL;
            END_VAR

            _runtimeParameters^.JogSpeed := value;
        END_METHOD

        METHOD PUBLIC SetJogHighSpeed
            VAR_INPUT
                value : LREAL;
            END_VAR

            _runtimeParameters^.JogHighSpeed := value;
        END_METHOD

        METHOD PUBLIC SetObjectRadius
            VAR_INPUT
                value : LREAL;
            END_VAR

            _runtimeParameters^.ObjectRadius := value;
        END_METHOD

        METHOD PUBLIC JogPositive
            VAR_INPUT
                highSpeed : BOOL := FALSE;
            END_VAR

            _jogUseHighSpeed := highSpeed;
            _jogPositive := TRUE;
        END_METHOD

        METHOD PUBLIC JogNegative
            VAR_INPUT
                highSpeed : BOOL := FALSE;
            END_VAR

            _jogUseHighSpeed := highSpeed;
            _jogNegative := TRUE;
        END_METHOD

        METHOD PUBLIC IsEnabled : BOOL
            IsEnabled := _axis.GetStatus().enable;
        END_METHOD

        METHOD PUBLIC IsBusy : BOOL
            IsBusy := FALSE;

            IF _latestCommand <> NULL THEN
                IsBusy := _latestCommand.Busy();
            ELSIF _latestHomingCommand <> NULL THEN
                IsBusy := _latestHomingCommand.Busy();
            END_IF;
        END_METHOD

        METHOD PUBLIC HasError : BOOL
            HasError := FALSE;

            IF _latestCommand <> NULL THEN
                HasError := _latestCommand.Error();
            ELSIF _latestHomingCommand <> NULL THEN
                HasError := _latestHomingCommand.Error();
            END_IF;
        END_METHOD

        METHOD PUBLIC AtStandstill : BOOL
            AtStandstill := _axis.GetStatus().standstill;
        END_METHOD

        METHOD PUBLIC IsHomed : BOOL
            IsHomed := _axis.GetStatus().homingDone;
        END_METHOD

        METHOD PUBLIC ActualLinearPosition : LREAL
            ActualLinearPosition := _axis.GetPositioningAxisRef()^.ActualPosition;
        END_METHOD

        METHOD PUBLIC ActualLinearVelocity : LREAL
            ActualLinearVelocity := _axis.GetPositioningAxisRef()^.ActualVelocity;
        END_METHOD

        METHOD PUBLIC ActualAngularPosition : LREAL
            ;
        END_METHOD

        METHOD PUBLIC ActualAngularVelocity : LREAL
            ;
        END_METHOD

        METHOD PUBLIC OVERRIDE Observe : IAssetObservable
            Observe := _observable;
        END_METHOD

        METHOD PRIVATE UpdateObservable
            _observable.Enabled := THIS.IsEnabled();
            _observable.Accelerating := FALSE; // TODO: Implement
            _observable.Decelerating := FALSE; // TODO: Implement
            _observable.Standstill := THIS.AtStandstill();
            _observable.Homed := THIS.IsHomed();
            _observable.Error := THIS.HasError();
            _observable.ErrorId := WORD#16#FFFF; // TODO: Implement
            _observable.Busy := THIS.IsBusy();
            _observable.Done := FALSE; // TODO: Implement
            _observable.LinearPosition := THIS.ActualLinearPosition();
            _observable.LinearVelocity := THIS.ActualLinearVelocity();
            _observable.LatestCommandId := -1; // TODO: Implement
        END_METHOD
    END_CLASS

END_NAMESPACE

(* ---- TechnologyObjects.st ---- *)
USING Siemens.Simatic.S71500.MotionControl;
USING Siemens.Simatic.S71500.MotionControl.Native;

NAMESPACE Esab.Motion

    CLASS TechnologyObjects
        VAR PRIVATE
            _horizontalSlideAxisDb : DB_ANY;
            _verticalSlideAxisDb : DB_ANY;

            _attached : BOOL := FALSE;
            _horizontalSlideAxisInstance : PosAxis;
            _verticalSlideAxisInstance : PosAxis;
        END_VAR

        METHOD PUBLIC Setup
            VAR_INPUT
                horizontalSlideAxisDb : DB_ANY;
                verticalSlideAxisDb : DB_ANY;
            END_VAR

            _horizontalSlideAxisDb := horizontalSlideAxisDb;
            _verticalSlideAxisDb := verticalSlideAxisDb;

            _attached :=  _horizontalSlideAxisInstance.Attach(_horizontalSlideAxisDb) AND _verticalSlideAxisInstance.Attach(_verticalSlideAxisDb);
        END_METHOD

        METHOD PUBLIC IsAttached : BOOL
            IsAttached := _attached;
        END_METHOD

        METHOD PUBLIC GetHorizontalSlideAxis : itfPosAxis
            GetHorizontalSlideAxis := _horizontalSlideAxisInstance;
        END_METHOD

        METHOD PUBLIC GetVerticalSlideAxis : itfPosAxis
            GetVerticalSlideAxis := _verticalSlideAxisInstance;
        END_METHOD
    END_CLASS

END_NAMESPACE
